PROGRAM Coordinate_System
VAR

END_VAR

// NETWORK 1

// NETWORK 2

END_PROGRAM

(* stored: Version 1.1.0.1, ProductVersion 3.1.4018.9
   POU Coordinate_System: Id {9b64fdf4-5383-4113-8a9b-2347dd86728b}, SpecialFunc None *)
